% RSLogix 500 project I2P JOB 9 TIPPY.RSS, saved by version 10.00.00.00 %
PROJECT "UNTITLED"    % processor: Bul.1763 MicroLogix 1100 Series B %

PROGRAM FILES
  LAD 2   5 rungs

DATA FILES
  O0 OUTPUT  4 elements
  I1 INPUT  6 elements
  S2 STATUS  66 elements
  B3 BINARY  1 elements
  T4 TIMER  1 elements
  C5 COUNTER  1 elements
  R6 CONTROL  1 elements
  N7 INTEGER  1 elements
  F8 FLOAT  1 elements

LADDER 2
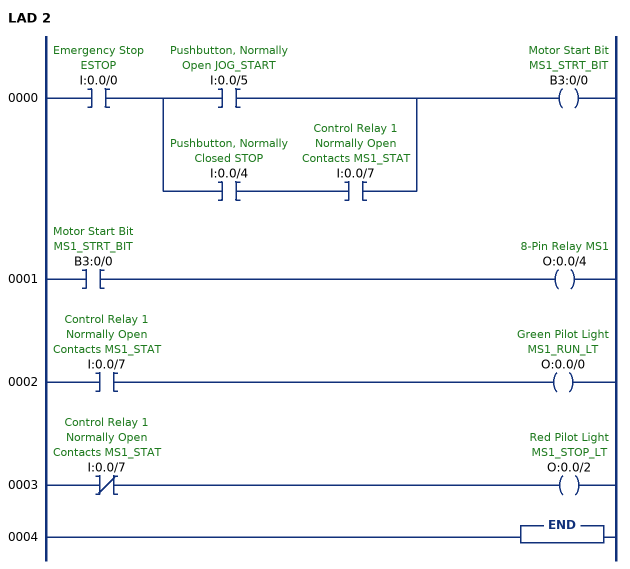
% Rung: 0 %
SOR XIC I:0.0/0 BST XIC I:0.0/5 NXB XIC I:0.0/4 XIC I:0.0/7 BND OTE B3:0/0 EOR
%   I:0.0/0  ESTOP  "Emergency Stop" %
%   I:0.0/5  JOG_START  "Pushbutton, Normally Open" %
%   I:0.0/4  STOP  "Pushbutton, Normally Closed" %
%   I:0.0/7  MS1_STAT  "Control Relay 1 Normally Open Contacts" %
%   B3:0/0  MS1_STRT_BIT  "Motor Start Bit" %
% Rung: 1 %
SOR XIC B3:0/0 OTE O:0.0/4 EOR
%   B3:0/0  MS1_STRT_BIT  "Motor Start Bit" %
%   O:0.0/4  MS1  "8-Pin Relay" %
% Rung: 2 %
SOR XIC I:0.0/7 OTE O:0.0/0 EOR
%   I:0.0/7  MS1_STAT  "Control Relay 1 Normally Open Contacts" %
%   O:0.0/0  MS1_RUN_LT  "Green Pilot Light" %
% Rung: 3 %
SOR XIO I:0.0/7 OTE O:0.0/2 EOR
%   I:0.0/7  MS1_STAT  "Control Relay 1 Normally Open Contacts" %
%   O:0.0/2  MS1_STOP_LT  "Red Pilot Light" %
% Rung: 4 %
SOR END EOR

OTHER DOCUMENTED ADDRESSES
  I:0.0/1  3PS_A  "3-Position Selector Switch Position A"
  I:0.0/2  3PS_B  "3-Position Selector Switch Position B"
  I:0.0/3  2PS_A  "2-Position Selector Switch"
  I:0.0/6  PB_NO_2  "Pushbutton, Normally Open"
  I:0.0/8  CR_NO_2  "Control Relay 2 Normaly Open Contacts"
  I:0.0/9  MS_REV  "Reverse Motor Starter Normally Open Contacts"
